FUNCTION F_UpdateUsingVAR : BOOL
VAR_IN_OUT
	nNumber1 : DINT;
END_VAR
VAR
END_VAR

nNumber1 := nNumber1 + 1;

END_FUNCTION

(* stored: Version 1.1.0.1, ProductVersion 3.1.4024.16
   POU F_UpdateUsingVAR: Id {8da0a965-50a0-413d-ac37-631c411fc1d5}, SpecialFunc None *)
